// TIA Portal V16 export
// export: Created 2024-08-24T20:12:49.1702239Z, ExportSetting WithDefaults, DisplayName Totally Integrated Automation Portal, DisplayVersion V16, DisplayName TIA Portal Version Control Interface, DisplayVersion V16, DisplayName TIA Portal Openness, DisplayVersion V16, DisplayName STEP 7 Professional, DisplayVersion V16, DisplayName STEP 7 Safety, DisplayVersion V16, DisplayName WinCC Professional, DisplayVersion V16
VAR_GLOBAL   // PLC tag table "Tabla de variables_1"
   entrada_io_1 AT %M11.0 : Bool;
   entrada_io_2 AT %M11.1 : Bool;
   entrada_io_3 AT %M11.2 : Bool;
   entrada_io_4 AT %M11.3 : Bool;
   entrada_io_5 AT %M11.4 : Bool;
   entrada_io_6 AT %M11.5 : Bool;
END_VAR
